FUNCTION_BLOCK CU010SuspendTask EXTENDS CUBaseSuspend IMPLEMENTS ICUTask
VAR

END_VAR

Run();

(*~
	<docu>
		<summary>
			Main method of the sequener. Custom code needs to be placed here. The sequencer is executed by call of **Instance.Run()** method.
			This method is abstract, and it must be overridden in derived block.
		</summary>
	</docu>
~*)
METHOD PROTECTED Main : BOOL
(*

	SUSPEND PROCESS 
	Following steps provide suspend actions for this controlled unit.
	Add components add write customized sequence according to your need.
*)

		
//
IF (Step(100, TRUE, '<#WAITING FOR START#>')) THEN
    //-------------------------------------    

    StepCompleteWhen(TRUE);
    //-------------------------------------
END_IF

//HERE  YOU CAN WRITE  WHAT IS NECESSARY 
//TO SUPSEND  PROCESS..... TO INTERUPT SAFETY

IF (Step(1000, TRUE, '<#SUSPENDING COMPONENTS#>')) THEN
 	//-------------------------------------    
	//StepCompleteWhen(Station.AutomatTask.CurrentStep.Status <> eStepStatus.Running);
		
    StepCompleteWhen( CurrentStep.Duration >= T#3000MS);
    //-------------------------------------
END_IF

IF (Step(30000, TRUE, 'SUSPEND DONE')) THEN
    //-------------------------------------
		
        THIS^._done:=TRUE;
		THIS^.Task.DoneWhen(TRUE);
	
   
    //-------------------------------------	
END_IF
END_METHOD

METHOD PUBLIC OnStart
SUPER^.OnStart();
Station.RecoverTask.Restore();
END_METHOD

PROPERTY Station : REFERENCE TO CU010
GET
VAR
    _station : POINTER TO CU010;
END_VAR
IF __QUERYPOINTER(Parent, _station) THEN // Check if _Parent is Station001
    Station REF= _station^;              // If the check is successful dereference a pointer. simlar to THIS^ or SUPER^
END_IF
END_GET
END_PROPERTY

END_FUNCTION_BLOCK

(* stored: Version 1.1.0.1
   POU CU010SuspendTask: Id {afedf12f-ca70-450e-8b3c-625c5da0a8a7}, SpecialFunc None
   Method Main: Id {0b06794c-bee3-42db-8f39-31d5a6d19c03}
   Method OnStart: Id {8a33d9a2-474c-4fff-9a6f-3b9e17fc0069}
   Property Station: Id {9ee83c1a-9f7d-41bc-8bbe-fc1dbd27ee12}
   Get Get: Id {4ca0ef88-fe4e-4127-bb27-7aa372f83574} *)
